// A string builder utility that allows for manipulation of a string up to 255 characters. It implements the I_Strb interface that allows for method chaining.
FUNCTION_BLOCK Strb IMPLEMENTS I_Strb
VAR
	_sString	: Str;
	_nLength	: INT;
END_VAR

PROPERTY PRIVATE _this : I_Strb
GET
VAR
	_iThis : I_Strb := THIS^;
END_VAR
_this := _iThis;
END_GET
END_PROPERTY

// Appends the specified string to the current string.
// Truncates if the total length exceeds 255 characters.
METHOD Append : I_Strb
VAR_INPUT
    sToAdd : Str; // String to append
END_VAR

VAR
	_nNewLength	: INT;
END_VAR
Append := _this;

IF sToAdd = '' THEN
	RETURN;
END_IF

_nNewLength := Tc2_Standard.LEN(sToAdd) + _nLength;
IF _nNewLength > 255 THEN
	_nNewLength := 255;
END_IF

_sString := Tc2_Standard.CONCAT(_sString, sToAdd);
_nLength := _nNewLength;
END_METHOD

// Finds the first occurrence of a substring after the specified position.
// Outputs the start and end positions of the found substring.
METHOD FindFirstAfter : I_Strb
VAR_INPUT
    sToFind : Str;      // Substring to find
    nPosition : INT := 1; // Starting position for search
END_VAR
VAR_OUTPUT
    nStart : INT;       // Start position of the found substring
    nEnd : INT;         // End position of the found substring
END_VAR

VAR
	_sTemp			: Str;
	_nOffset		: INT;
END_VAR
FindFirstAfter := _this;

IF sToFind = '' THEN
	RETURN;
END_IF

IF nPosition = 0 THEN
	RETURN;
END_IF

_sTemp := Tc2_Standard.MID(_sString, _nLength, nPosition);
IF (_nOffset := Tc2_Standard.FIND(_sTemp, sToFind)) <> 0 THEN
	nStart := nPosition + _nOffset - 1;
	nEnd := nPosition + _nOffset - 2 + Tc2_Standard.LEN(sToFind);
END_IF
END_METHOD

// Finds the last occurrence of a substring before the specified position.
// Outputs the start and end positions of the found substring.
METHOD FindLastBefore : I_Strb
VAR_INPUT
    sToFind : Str;        // Substring to find
    nPosition : INT := 256; // Starting position for reverse search
END_VAR
VAR_OUTPUT
    nStart : INT;         // Start position of the found substring
    nEnd : INT;           // End position of the found substring
END_VAR
VAR
	_sTemp			: Str;
	_nFindLength	: INT := Tc2_Standard.LEN(sToFind);
	_nOffset		: INT;
END_VAR
FindLastBefore := _this;

IF sToFind = '' THEN
	RETURN;
END_IF

IF nPosition = 0 THEN
	RETURN;
END_IF

IF nPosition = 256 THEN
	nPosition := _nLength;
END_IF

REPEAT
	_sTemp := Tc2_Standard.MID(_sString, _nFindLength, nPosition);
	IF _sTemp = sToFind THEN
		nStart 	:= nPosition;
		nEnd	:= nPosition + _nFindLength - 1;
		RETURN;
	END_IF
UNTIL
	(nPosition := nPosition - 1) <= 0
END_REPEAT
END_METHOD

// Checks if the specified substring exists after the given position.
METHOD HasAfter : BOOL
VAR_INPUT
    sToFind : Str;      // Substring to search for
    nPosition : INT := 0; // Starting position for search
END_VAR
VAR_OUTPUT
    nStart : INT;       // Start position of the found substring
    nEnd : INT;         // End position of the found substring
END_VAR
FindFirstAfter(sToFind, nPosition, nStart => nStart, nEnd => nEnd);
HasAfter := nStart > 0;
END_METHOD

// Checks if the specified substring exists before the given position.
METHOD HasBefore : BOOL
VAR_INPUT
    sToFind : Str;        // Substring to search for
    nPosition : INT := 256; // Ending position for reverse search
END_VAR
VAR_OUTPUT
    nStart : INT;         // Start position of the found substring
    nEnd : INT;           // End position of the found substring
END_VAR
IF nPosition = 256 THEN
	nPosition := Tc2_Standard.LEN(_sString);
END_IF

FindLastBefore(sToFind, nPosition, nStart => nStart, nEnd => nEnd);
HasBefore := nStart > 0;
END_METHOD

// Inserts a specified substring at a given position.
// Truncates if the total length exceeds 255 characters.
METHOD Inject : I_Strb
VAR_INPUT
    nPosition : INT;    // Position to inject the string
    sToInject : Str;    // String to inject
END_VAR
VAR
	_nNewLength	: INT;
END_VAR
Inject := _this;

IF sToInject = '' THEN
	RETURN;
END_IF

IF nPosition = 0 THEN
	RETURN;
END_IF

IF nPosition > _nLength THEN
	RETURN;
END_IF

_nNewLength := Tc2_Standard.LEN(sToInject) + _nLength;
IF _nNewLength > 255 THEN
	_nNewLength := 255;
END_IF

_sString := Tc2_Standard.INSERT(_sString, sToInject, nPosition);
_nLength := _nNewLength;
END_METHOD

// Checks if the current string is empty.
METHOD IsEmpty : BOOL
VAR_INPUT
END_VAR
IsEmpty := _nLength = 0;
END_METHOD

// Returns the current length of the string.
// The length of the string is stored as a separate variable (_nLength) 
// and reflects the actual length of the content.
// Unlike Tc2_Standard.LEN(), which counts up to the first null character, 
// this method directly returns the stored length.
METHOD Length : INT
VAR_INPUT
END_VAR
Length := _nLength;
END_METHOD

// Prepends the specified string to the current string.
// Truncates if the total length exceeds 255 characters.
METHOD Prepend : I_Strb
VAR_INPUT
    sToAdd : Str; // String to prepend
END_VAR
VAR
	_nNewLength	: INT;
END_VAR
Prepend := _this;

IF sToAdd = '' THEN
	RETURN;
END_IF

_nNewLength := Tc2_Standard.LEN(sToAdd) + _nLength;
IF _nNewLength > 255 THEN
	_nNewLength := 255;
END_IF

_sString := Tc2_Standard.CONCAT(sToAdd, _sString);
_nLength := _nNewLength;
END_METHOD

// Returns the current string value.
METHOD Read : Str
VAR_INPUT
END_VAR
Read := _sString;
END_METHOD

// Removes a substring of specified length starting at a given position.
METHOD Remove : I_Strb
VAR_INPUT
    nLength : INT;    // Length of the substring to remove
    nPosition : INT;  // Starting position of the substring to remove
END_VAR

VAR
	_nPosition	: INT;
END_VAR
Remove := _this;

IF nPosition = 0 THEN
	RETURN;
END_IF

IF nPosition > _nLength THEN
	RETURN;
END_IF

IF nLength = 0 THEN
	RETURN;
END_IF

IF nLength + nPosition > _nLength THEN
	nLength := _nLength - nPosition + 1;
END_IF

_sString := Tc2_Standard.DELETE(_sString, nLength, nPosition);
_nLength := _nLength - nLength;
END_METHOD

// Sets the current string to a new value.
METHOD Set : I_Strb
VAR_INPUT
    sLiteral : Str; // New string value
END_VAR
Set 		:= _this;

_sString 	:= sLiteral;
_nLength	:= Tc2_Standard.LEN(sLiteral);
END_METHOD

// Extracts a substring starting from a given position with a specified length.
METHOD Slice : I_Strb
VAR_INPUT
    nPosition : INT; // Starting position of the slice
    nLength : INT;   // Length of the slice
END_VAR
VAR_OUTPUT
    sSlice : Strb;   // The sliced string
END_VAR
Slice := _this;

IF nPosition = 0 THEN
	RETURN;
END_IF

IF nLength = 0 THEN
	RETURN;
END_IF

sSlice.Set(Tc2_Standard.MID(_sString, nLength, nPosition));
END_METHOD

// Splits the string into two parts at the specified position.
METHOD Split : I_Strb
VAR_INPUT
    nPosition : INT; // Position to split the string
END_VAR
VAR_OUTPUT
    sLeft : Strb;    // Left part of the split
    sRight : Strb;   // Right part of the split
END_VAR
Split := _this;

IF nPosition = 0 THEN
	RETURN;
END_IF

sLeft.Set(Tc2_Standard.LEFT(_sString, nPosition));
sRight.Set(Tc2_Standard.RIGHT(_sString, _nLength - nPosition));
END_METHOD

END_FUNCTION_BLOCK

(* stored: Version 1.1.0.1
   POU Strb: Id {097a9ce5-fff4-459c-bf61-90e104e444f4}, SpecialFunc None
   Folder _: Id {ee5226c4-1bfb-4c78-b582-ae1ec7e3d151}
   Folder I_Build: Id {ac6c8744-50a3-4f05-8763-d0edced1682d}
   Property _this: Id {9f5d4af9-6657-4b84-b94c-f143552d6daa}
   Get Get: Id {57c7bcd7-c66a-4ed8-9ead-784876349f3a}
   Method Append: Id {7f7905f2-7818-4e4d-8188-6df497128569}
   Method FindFirstAfter: Id {8f9e101f-7a2f-44e6-8d32-11ba6ad80cd3}
   Method FindLastBefore: Id {71bc0f49-5ad9-4169-b5ad-3a872c3c466c}
   Method HasAfter: Id {f544f3ca-8838-4319-9707-f592713024e1}
   Method HasBefore: Id {62915ef4-82cd-46dc-8a4f-63e40918902b}
   Method Inject: Id {2e9ce33a-9a18-4428-92c8-44eae0f3e5ac}
   Method IsEmpty: Id {56f58905-f285-454e-bc54-bf4b7769c906}
   Method Length: Id {bd663ea8-cc03-4934-83d1-a6fc1b5f2021}
   Method Prepend: Id {90cd07b0-8292-43be-8f7c-ccc1f2a79b9d}
   Method Read: Id {201b7f18-5c0a-4280-87a7-27b4592e313f}
   Method Remove: Id {87c2b449-3936-4b9e-bf9e-9a7e13244b52}
   Method Set: Id {4e083d1b-9de2-4451-b0f9-5b881e2173d3}
   Method Slice: Id {41b26e98-f082-480a-832d-cfbb05d20b83}
   Method Split: Id {8062e340-a176-420f-bbf7-07ca296bea0b} *)
